TYPE ST_ITC_SubsystemCommandsEmulation :
(**************************************************************************************
 * 	Application		:	BoxControl Framework
 *	Revision		:	$Revision: 404529 $
 *	Revision date	:	$Date: 2018-04-23 08:21:38 +0200 (Mo., 23 Apr 2018) $
 *	Last changed by	:	$Author: b7bolm $
 *	URL				:	$URL: http://almscdc.swisslog.com/repo/SWPD/Development/BoxControlFramework/20_Release/trunk/01_Software/BCF/BCF/JumpStart/20_Product/11_Emu/15_Subsystem/10_Lib/10_Conv/01_DUTs/ST_ITC_SubSystemCommandsEmulation.TcDUT $
 *
 *	Purpose			:	Subsystem ITC commands emulation
 *
 * ------------------------------------------------------------------------------------
 *	Copyright Swisslog [IP AG], Switzerland. All rights reserved.
 * 
 * ------------------------------------------------------------------------------------
 *	
 * 	Revision History: 
 *
 * 	VERSION			DATE			INITIALS			DESCRIPTION
 *	0.1				01.01.2001		swl					Example
 *
 **************************************************************************************)
STRUCT
	Error				: BOOL; // Command to set and reset an error
	ErrorCode			: INT;  // ErrorCode for the error which has to be produced
END_STRUCT
END_TYPE

(* stored: Version 1.1.0.1, ProductVersion 3.1.4022.12
   DUT ST_ITC_SubSystemCommandsEmulation: Id {920b6266-0451-44e4-b6be-1d7db1c3d0d8} *)
